INTERFACE I_ChunkedRequestsManager

METHOD PUBLIC TryHandleIncomingRequest : BOOL
VAR_INPUT
	Request : I_Request;
	Response : I_ServerResponse;
	NextMidleware : I_Middleware;
END_VAR
END_METHOD

END_INTERFACE

(* stored: Version 1.1.0.1, ProductVersion 3.1.4026.13
   Itf I_ChunkedRequestsManager: Id {9239929f-223e-4c1e-9172-63a672c2a44f}
   Method TryHandleIncomingRequest: Id {4efc3b08-734c-4b9b-a14e-d531293f1584} *)
